// Mitsubishi GX Works2 project: 자동   PLC: Q02/Q02H

PROGRAM MAIN
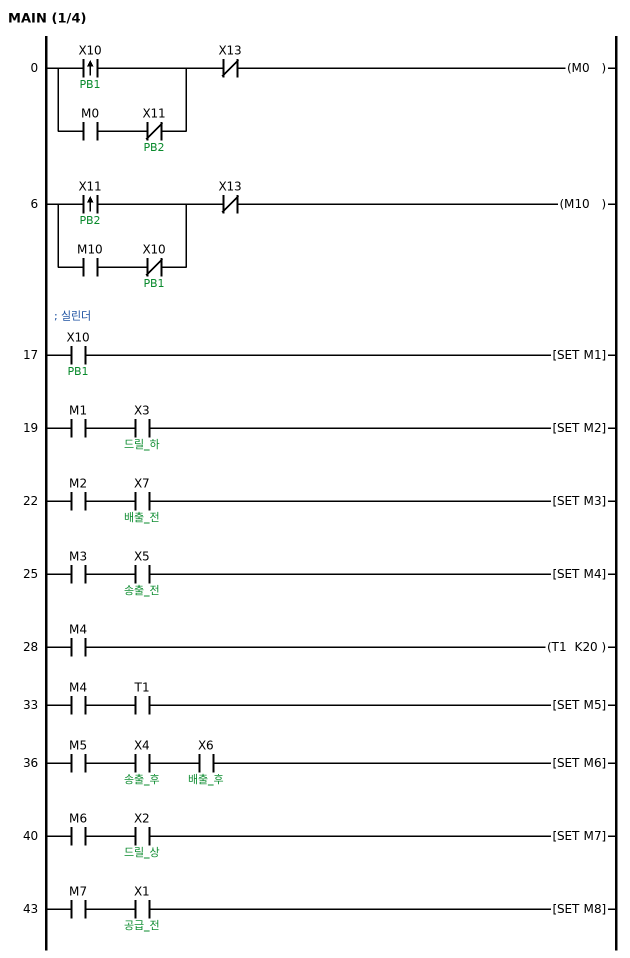
0     LDP     X10  ; PB1
      LD      M0
      ANI     X11  ; PB2
      ORB
      ANI     X13
      OUT     M0
6     LDP     X11  ; PB2
      LD      M10
      ANI     X10  ; PB1
      ORB
      ANI     X13
      OUT     M10
; 실린더
17    LD      X10  ; PB1
      SET     M1
19    LD      M1
      AND     X3  ; 드릴_하
      SET     M2
22    LD      M2
      AND     X7  ; 배출_전
      SET     M3
25    LD      M3
      AND     X5  ; 송출_전
      SET     M4
28    LD      M4
      OUT     T1 K20
33    LD      M4
      AND     T1
      SET     M5
36    LD      M5
      AND     X4  ; 송출_후
      AND     X6  ; 배출_후
      SET     M6
40    LD      M6
      AND     X2  ; 드릴_상
      SET     M7
43    LD      M7
      AND     X1  ; 공급_전
      SET     M8
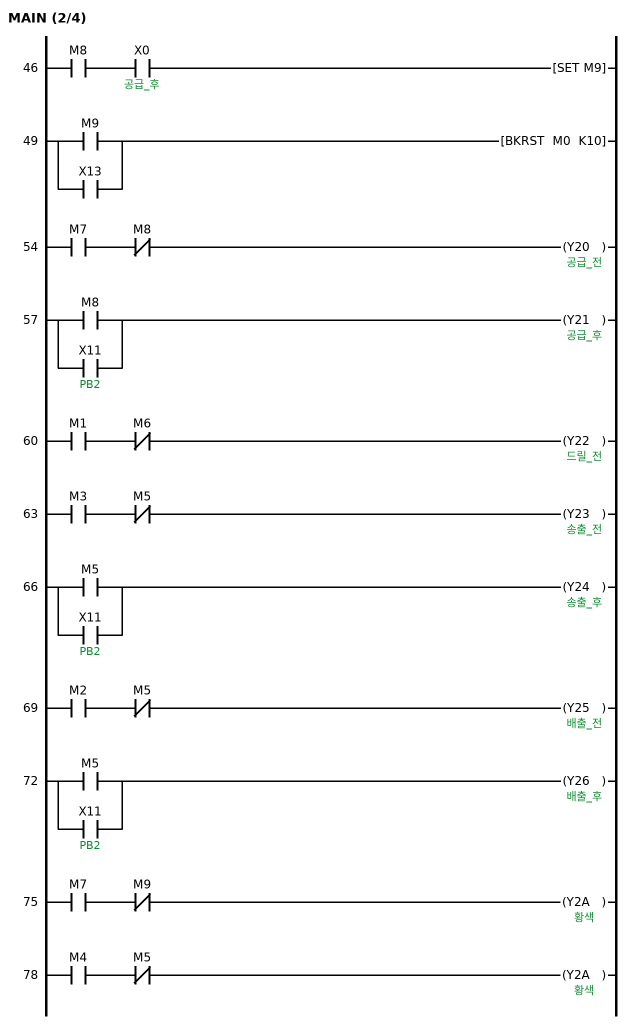
46    LD      M8
      AND     X0  ; 공급_후
      SET     M9
49    LD      M9
      OR      X13
      BKRST   M0 K10
54    LD      M7
      ANI     M8
      OUT     Y20  ; 공급_전
57    LD      M8
      OR      X11  ; PB2
      OUT     Y21  ; 공급_후
60    LD      M1
      ANI     M6
      OUT     Y22  ; 드릴_전
63    LD      M3
      ANI     M5
      OUT     Y23  ; 송출_전
66    LD      M5
      OR      X11  ; PB2
      OUT     Y24  ; 송출_후
69    LD      M2
      ANI     M5
      OUT     Y25  ; 배출_전
72    LD      M5
      OR      X11  ; PB2
      OUT     Y26  ; 배출_후
75    LD      M7
      ANI     M9
      OUT     Y2A  ; 황색
78    LD      M4
      ANI     M5
      OUT     Y2A  ; 황색
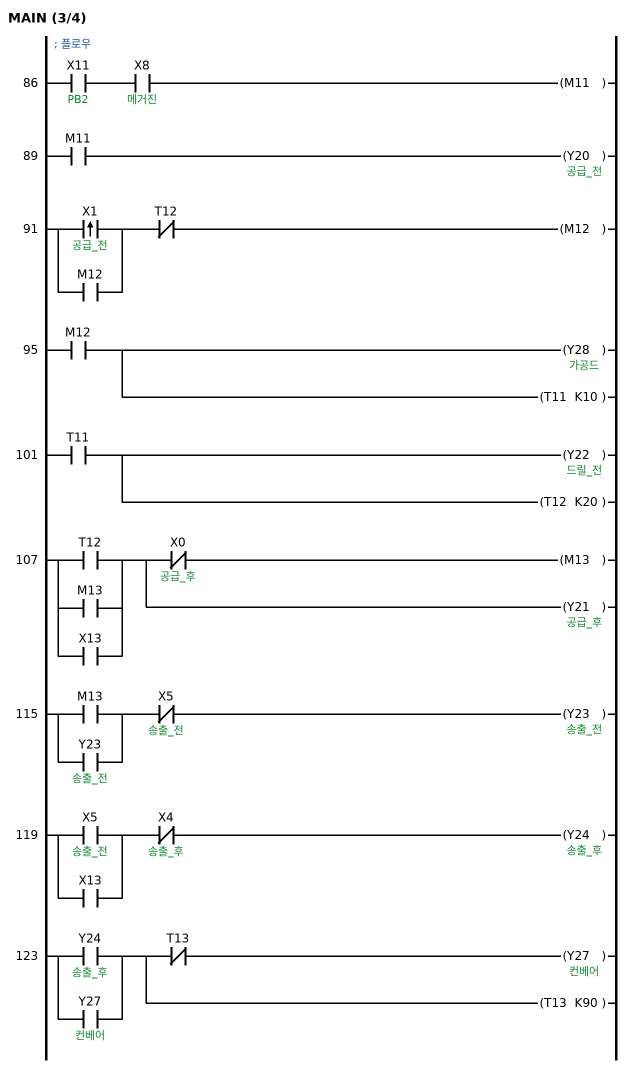
; 플로우
86    LD      X11  ; PB2
      AND     X8  ; 메거진
      OUT     M11
89    LD      M11
      OUT     Y20  ; 공급_전
91    LDP     X1  ; 공급_전
      OR      M12
      ANI     T12
      OUT     M12
95    LD      M12
      OUT     Y28  ; 가공드
      OUT     T11 K10
101   LD      T11
      OUT     Y22  ; 드릴_전
      OUT     T12 K20
107   LD      T12
      OR      M13
      OR      X13
      MPS
      ANI     X0  ; 공급_후
      OUT     M13
      MPP
      OUT     Y21  ; 공급_후
115   LD      M13
      OR      Y23  ; 송출_전
      ANI     X5  ; 송출_전
      OUT     Y23  ; 송출_전
119   LD      X5  ; 송출_전
      OR      X13
      ANI     X4  ; 송출_후
      OUT     Y24  ; 송출_후
123   LD      Y24  ; 송출_후
      OR      Y27  ; 컨베어
      MPS
      ANI     T13
      OUT     Y27  ; 컨베어
      MPP
      OUT     T13 K90
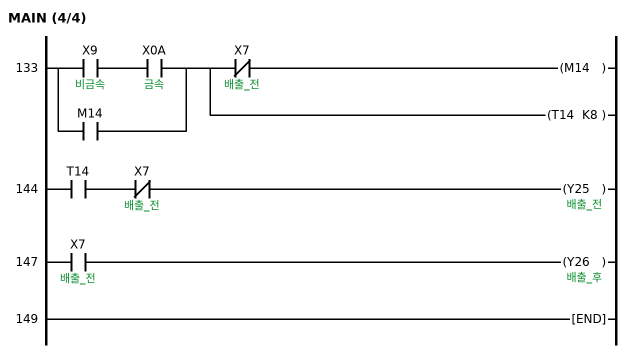
133   LD      X9  ; 비금속
      AND     X0A  ; 금속
      OR      M14
      MPS
      ANI     X7  ; 배출_전
      OUT     M14
      MPP
      OUT     T14 K8
144   LD      T14
      ANI     X7  ; 배출_전
      OUT     Y25  ; 배출_전
147   LD      X7  ; 배출_전
      OUT     Y26  ; 배출_후
149   END
END_PROGRAM

// device comments not shown above
X12  ; PB3
Y29  ; 적색
Y2B  ; 녹색
